FUNCTION "FC 141" : VOID	// FC 141
VERSION : 0.1
BEGIN
// (block stored without names or comments; labels and parameter names are numbered)
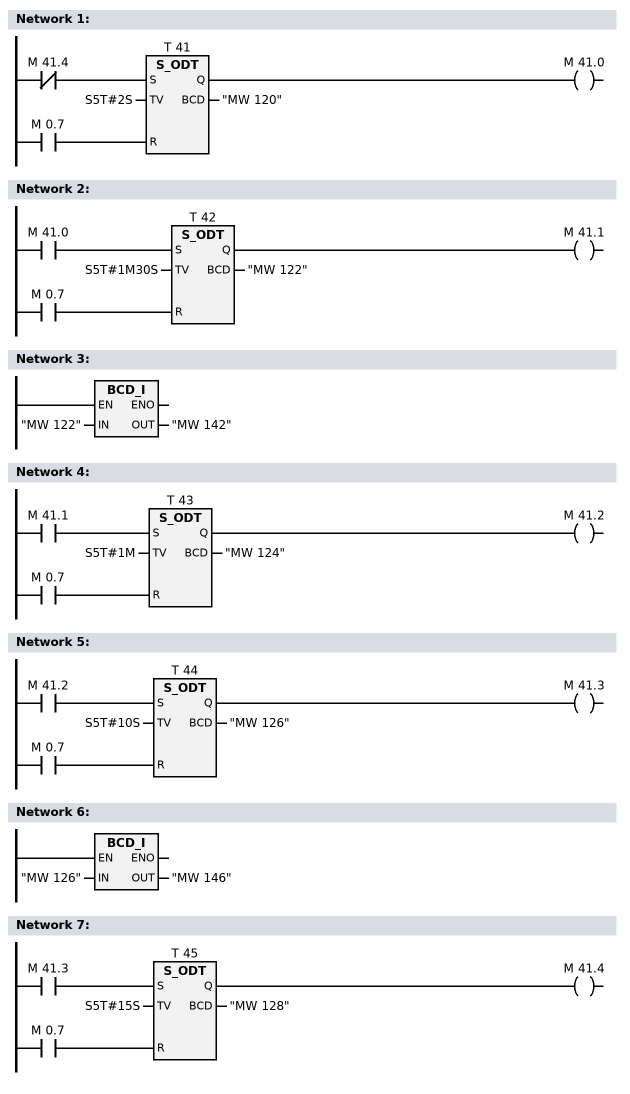
NETWORK
TITLE =
      AN    "M 41.4";
      L     S5T#2S;
      SD    "T 41";
      A     "M 0.7";
      R     "T 41";
      NOP   0;
      LC    "T 41";
      T     "MW 120";
      A     "T 41";
      =     "M 41.0";
NETWORK
TITLE =
      A     "M 41.0";
      L     S5T#1M30S;
      SD    "T 42";
      A     "M 0.7";
      R     "T 42";
      NOP   0;
      LC    "T 42";
      T     "MW 122";
      A     "T 42";
      =     "M 41.1";
NETWORK
TITLE =
      L     "MW 122";
      BTI;
      T     "MW 142";
      NOP   0;
NETWORK
TITLE =
      A     "M 41.1";
      L     S5T#1M;
      SD    "T 43";
      A     "M 0.7";
      R     "T 43";
      NOP   0;
      LC    "T 43";
      T     "MW 124";
      A     "T 43";
      =     "M 41.2";
NETWORK
TITLE =
      A     "M 41.2";
      L     S5T#10S;
      SD    "T 44";
      A     "M 0.7";
      R     "T 44";
      NOP   0;
      LC    "T 44";
      T     "MW 126";
      A     "T 44";
      =     "M 41.3";
NETWORK
TITLE =
      L     "MW 126";
      BTI;
      T     "MW 146";
      NOP   0;
NETWORK
TITLE =
      A     "M 41.3";
      L     S5T#15S;
      SD    "T 45";
      A     "M 0.7";
      R     "T 45";
      NOP   0;
      LC    "T 45";
      T     "MW 128";
      A     "T 45";
      =     "M 41.4";
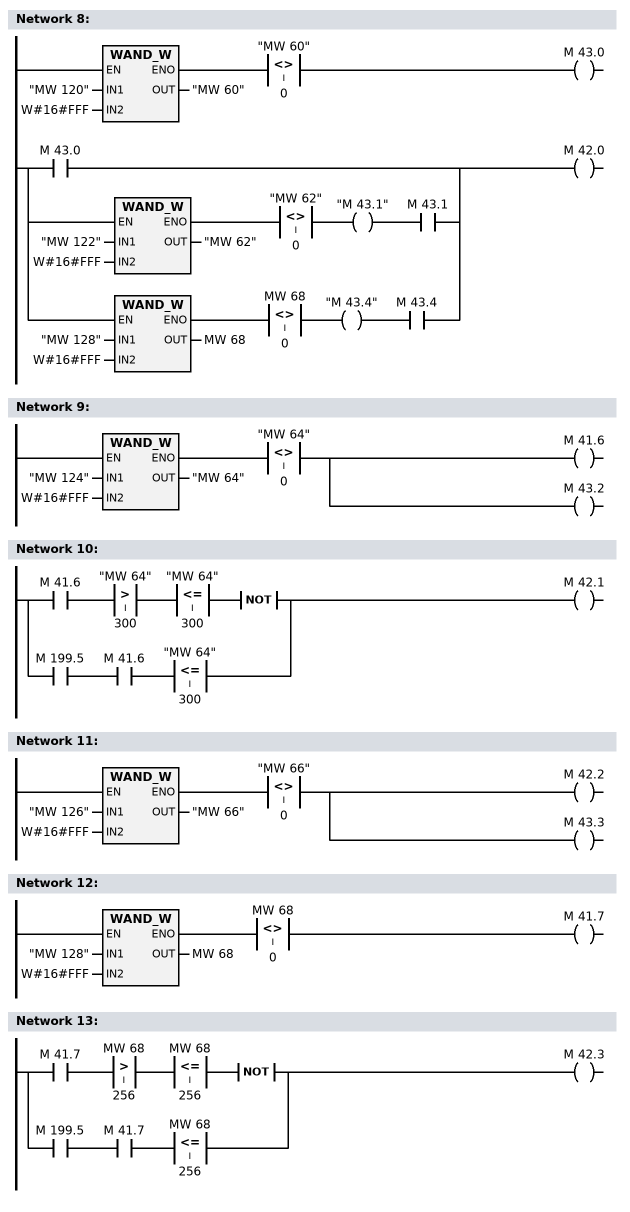
NETWORK
TITLE =
      A(;
      L     "MW 120";
      L     W#16#FFF;
      AW;
      T     "MW 60";
      SET;
      SAVE;
      CLR;
      A     BR;
      );
      A(;
      L     "MW 60";
      L     0;
      <>I;
      );
      =     "M 43.0";
      A     "M 43.0";
      O(;
      A(;
      L     "MW 122";
      L     W#16#FFF;
      AW;
      T     "MW 62";
      SET;
      SAVE;
      CLR;
      A     BR;
      );
      A(;
      L     "MW 62";
      L     0;
      <>I;
      );
      =     "M 43.1";
      A     "M 43.1";
      );
      O(;
      A(;
      L     "MW 128";
      L     W#16#FFF;
      AW;
      T     MW 68;
      SET;
      SAVE;
      CLR;
      A     BR;
      );
      A(;
      L     MW 68;
      L     0;
      <>I;
      );
      =     "M 43.4";
      A     "M 43.4";
      );
      =     "M 42.0";
NETWORK
TITLE =
      A(;
      L     "MW 124";
      L     W#16#FFF;
      AW;
      T     "MW 64";
      SET;
      SAVE;
      CLR;
      A     BR;
      );
      A(;
      L     "MW 64";
      L     0;
      <>I;
      );
      =     "M 41.6";
      =     "M 43.2";
NETWORK
TITLE =
      A     "M 41.6";
      A(;
      L     "MW 64";
      L     300;
      >I;
      );
      A(;
      A(;
      L     "MW 64";
      L     300;
      <=I;
      );
      NOT;
      );
      O;
      A     "M 199.5";
      A     "M 41.6";
      A(;
      L     "MW 64";
      L     300;
      <=I;
      );
      =     "M 42.1";
NETWORK
TITLE =
      A(;
      L     "MW 126";
      L     W#16#FFF;
      AW;
      T     "MW 66";
      SET;
      SAVE;
      CLR;
      A     BR;
      );
      A(;
      L     "MW 66";
      L     0;
      <>I;
      );
      =     "M 42.2";
      =     "M 43.3";
NETWORK
TITLE =
      A(;
      L     "MW 128";
      L     W#16#FFF;
      AW;
      T     MW 68;
      SET;
      SAVE;
      CLR;
      A     BR;
      );
      A(;
      L     MW 68;
      L     0;
      <>I;
      );
      =     "M 41.7";
NETWORK
TITLE =
      A     "M 41.7";
      A(;
      L     MW 68;
      L     256;
      >I;
      );
      A(;
      A(;
      L     MW 68;
      L     256;
      <=I;
      );
      NOT;
      );
      O;
      A     "M 199.5";
      A     "M 41.7";
      A(;
      L     MW 68;
      L     256;
      <=I;
      );
      =     "M 42.3";
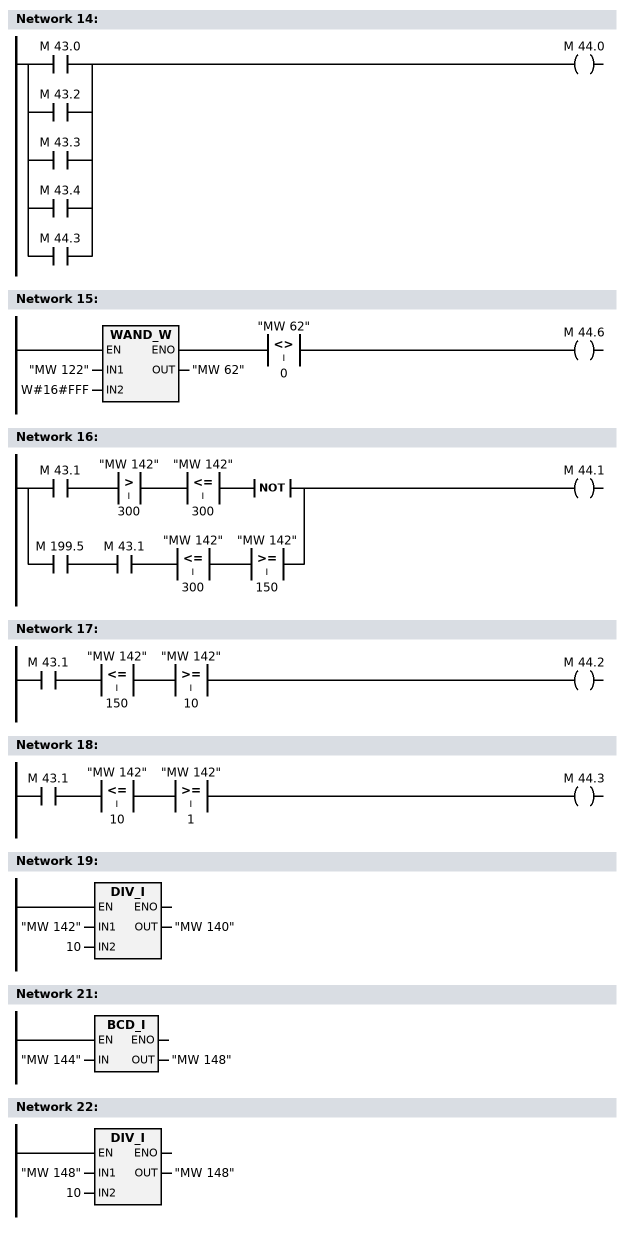
NETWORK
TITLE =
      O     "M 43.0";
      O     "M 43.2";
      O     "M 43.3";
      O     "M 43.4";
      O     M 44.3;
      =     "M 44.0";
NETWORK
TITLE =
      A(;
      L     "MW 122";
      L     W#16#FFF;
      AW;
      T     "MW 62";
      SET;
      SAVE;
      CLR;
      A     BR;
      );
      A(;
      L     "MW 62";
      L     0;
      <>I;
      );
      =     "M 44.6";
NETWORK
TITLE =
      A     "M 43.1";
      A(;
      L     "MW 142";
      L     300;
      >I;
      );
      A(;
      A(;
      L     "MW 142";
      L     300;
      <=I;
      );
      NOT;
      );
      O;
      A     "M 199.5";
      A     "M 43.1";
      A(;
      L     "MW 142";
      L     300;
      <=I;
      );
      A(;
      L     "MW 142";
      L     150;
      >=I;
      );
      =     "M 44.1";
NETWORK
TITLE =
      A     "M 43.1";
      A(;
      L     "MW 142";
      L     150;
      <=I;
      );
      A(;
      L     "MW 142";
      L     10;
      >=I;
      );
      =     "M 44.2";
NETWORK
TITLE =
      A     "M 43.1";
      A(;
      L     "MW 142";
      L     10;
      <=I;
      );
      A(;
      L     "MW 142";
      L     1;
      >=I;
      );
      =     M 44.3;
NETWORK
TITLE =
      L     "MW 142";
      L     10;
      /I;
      T     "MW 140";
      NOP   0;
NETWORK
TITLE =
      A(;
      A     "M 44.0";
      S     M 43.7;
      A     M 44.3;
      R     M 43.7;
      A     M 43.7;
      );
      L     S5T#1M10S;
      SD    "T 46";
      NOP   0;
      NOP   0;
      LC    "T 46";
      T     "MW 144";
      NOP   0;
NETWORK
TITLE =
      L     "MW 144";
      BTI;
      T     "MW 148";
      NOP   0;
NETWORK
TITLE =
      L     "MW 148";
      L     10;
      /I;
      T     "MW 148";
      NOP   0;
END_FUNCTION

FUNCTION "FC 142" : VOID	// FC 142
VERSION : 0.1
BEGIN
// (block stored without names or comments; labels and parameter names are numbered)
NETWORK
TITLE =
      A     "M 139.0";
      A     "M 139.1";
      CU    "Z 100";
      BLD   101;
      NOP   0;
      NOP   0;
      A(;
      L     "MW 150";
      L     60;
      >=I;
      );
      R     "Z 100";
      NOP   0;
      LC    "Z 100";
      T     "MW 160";
      NOP   0;
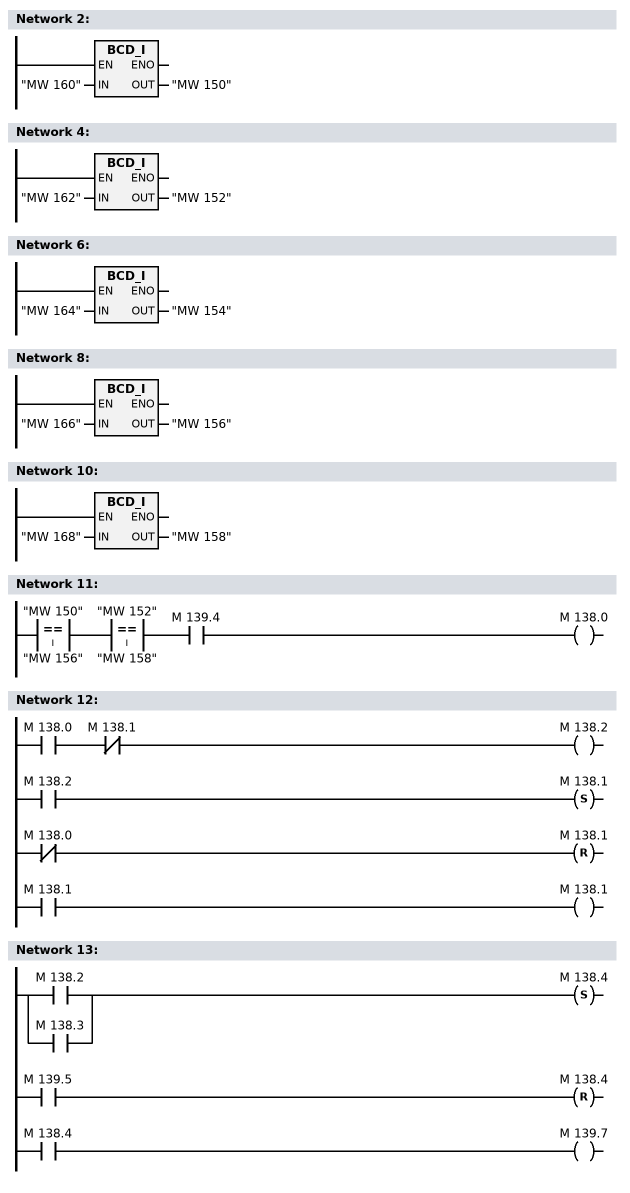
NETWORK
TITLE =
      L     "MW 160";
      BTI;
      T     "MW 150";
      NOP   0;
NETWORK
TITLE =
      A     "M 139.0";
      A     "M 139.2";
      CU    "Z 101";
      BLD   101;
      NOP   0;
      NOP   0;
      A(;
      L     "MW 152";
      L     24;
      >=I;
      );
      R     "Z 101";
      NOP   0;
      LC    "Z 101";
      T     "MW 162";
      NOP   0;
NETWORK
TITLE =
      L     "MW 162";
      BTI;
      T     "MW 152";
      NOP   0;
NETWORK
TITLE =
      A     "M 199.5";
      CU    "Z 102";
      BLD   101;
      NOP   0;
      NOP   0;
      A(;
      L     "MW 154";
      L     60;
      >=I;
      );
      R     "Z 102";
      NOP   0;
      LC    "Z 102";
      T     "MW 164";
      NOP   0;
NETWORK
TITLE =
      L     "MW 164";
      BTI;
      T     "MW 154";
      NOP   0;
NETWORK
TITLE =
      A(;
      A     "M 139.3";
      A     "M 139.1";
      O;
      A(;
      L     "MW 154";
      L     60;
      >=I;
      );
      AN    "M 139.3";
      );
      CU    "Z 103";
      BLD   101;
      NOP   0;
      NOP   0;
      A(;
      L     "MW 156";
      L     60;
      >=I;
      );
      R     "Z 103";
      NOP   0;
      LC    "Z 103";
      T     "MW 166";
      NOP   0;
NETWORK
TITLE =
      L     "MW 166";
      BTI;
      T     "MW 156";
      NOP   0;
NETWORK
TITLE =
      A(;
      A     "M 139.3";
      A     "M 139.2";
      O;
      A(;
      L     "MW 156";
      L     60;
      >=I;
      );
      AN    "M 139.3";
      );
      CU    "Z 104";
      BLD   101;
      NOP   0;
      NOP   0;
      A(;
      L     "MW 158";
      L     24;
      >=I;
      );
      R     "Z 104";
      NOP   0;
      LC    "Z 104";
      T     "MW 168";
      NOP   0;
NETWORK
TITLE =
      L     "MW 168";
      BTI;
      T     "MW 158";
      NOP   0;
NETWORK
TITLE =
      A(;
      L     "MW 150";
      L     "MW 156";
      ==I;
      );
      A(;
      L     "MW 152";
      L     "MW 158";
      ==I;
      );
      A     "M 139.4";
      =     "M 138.0";
NETWORK
TITLE =
      A     "M 138.0";
      AN    "M 138.1";
      =     "M 138.2";
      A     "M 138.2";
      S     "M 138.1";
      AN    "M 138.0";
      R     "M 138.1";
      A     "M 138.1";
      =     "M 138.1";
NETWORK
TITLE =
      A(;
      O     "M 138.2";
      O     "M 138.3";
      );
      S     "M 138.4";
      A     "M 139.5";
      R     "M 138.4";
      A     "M 138.4";
      =     "M 139.7";
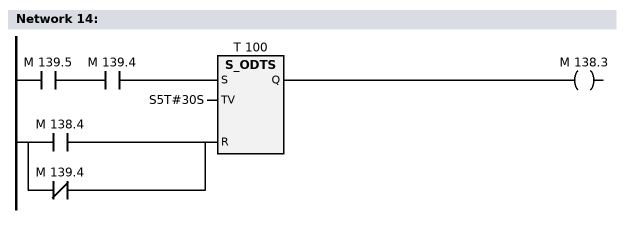
NETWORK
TITLE =
      A     "M 139.5";
      A     "M 139.4";
      L     S5T#30S;
      SS    "T 100";
      A(;
      O     "M 138.4";
      ON    "M 139.4";
      );
      R     "T 100";
      NOP   0;
      NOP   0;
      A     "T 100";
      =     "M 138.3";
END_FUNCTION

FUNCTION "FC 143" : VOID	// FC 143
VERSION : 0.1
BEGIN
// (block stored without names or comments; labels and parameter names are numbered)
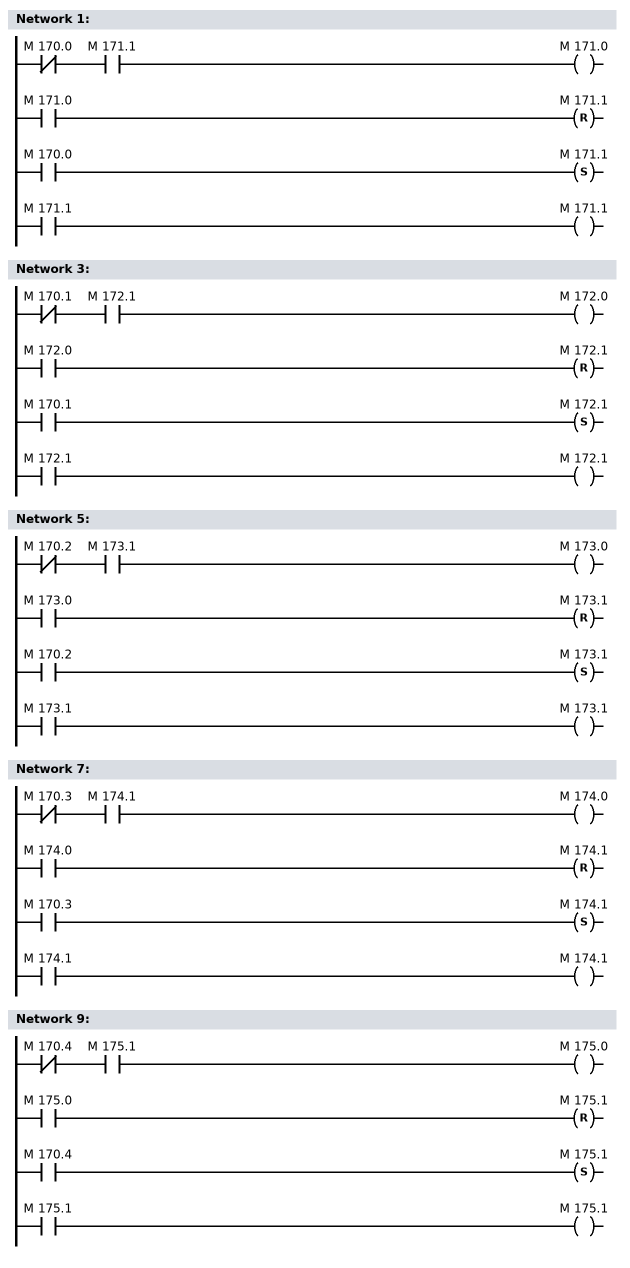
NETWORK
TITLE =
      AN    "M 170.0";
      A     "M 171.1";
      =     "M 171.0";
      A     "M 171.0";
      R     "M 171.1";
      A     "M 170.0";
      S     "M 171.1";
      A     "M 171.1";
      =     "M 171.1";
NETWORK
TITLE =
      A(;
      A     "M 171.0";
      S     "M 171.2";
      A     "M 190.1";
      R     "M 171.2";
      A     "M 171.2";
      );
      A     "M 1.5";
      O;
      AN    "M 171.2";
      A(;
      A     "M 171.0";
      S     "M 171.3";
      A     "M 190.2";
      A     "M 170.0";
      R     "M 171.3";
      A     "M 171.3";
      );
      O     "M 190.3";
      =     "M 171.4";
      =     "1H1";
NETWORK
TITLE =
      AN    "M 170.1";
      A     "M 172.1";
      =     "M 172.0";
      A     "M 172.0";
      R     "M 172.1";
      A     "M 170.1";
      S     "M 172.1";
      A     "M 172.1";
      =     "M 172.1";
NETWORK
TITLE =
      A(;
      A     "M 172.0";
      S     "M 172.2";
      A     "M 190.1";
      R     "M 172.2";
      A     "M 172.2";
      );
      A     "M 1.5";
      O;
      AN    "M 172.2";
      A(;
      A     "M 172.0";
      S     "M 172.3";
      A     "M 190.2";
      A     "M 170.1";
      R     "M 172.3";
      A     "M 172.3";
      );
      O     "M 190.3";
      =     "M 172.4";
      =     "2H1";
NETWORK
TITLE =
      AN    "M 170.2";
      A     "M 173.1";
      =     "M 173.0";
      A     "M 173.0";
      R     "M 173.1";
      A     "M 170.2";
      S     "M 173.1";
      A     "M 173.1";
      =     "M 173.1";
NETWORK
TITLE =
      A(;
      A     "M 173.0";
      S     "M 173.2";
      A     "M 190.1";
      R     "M 173.2";
      A     "M 173.2";
      );
      A     "M 1.5";
      O;
      AN    "M 173.2";
      A(;
      A     "M 173.0";
      S     "M 173.3";
      A     "M 190.2";
      A     "M 170.2";
      R     "M 173.3";
      A     "M 173.3";
      );
      O     "M 190.3";
      =     "M 173.4";
      =     "3H1";
NETWORK
TITLE =
      AN    "M 170.3";
      A     "M 174.1";
      =     "M 174.0";
      A     "M 174.0";
      R     "M 174.1";
      A     "M 170.3";
      S     "M 174.1";
      A     "M 174.1";
      =     "M 174.1";
NETWORK
TITLE =
      A(;
      A     "M 174.0";
      S     "M 174.2";
      A     "M 190.1";
      R     "M 174.2";
      A     "M 174.2";
      );
      A     "M 1.5";
      O;
      AN    "M 174.2";
      A(;
      A     "M 174.0";
      S     "M 174.3";
      A     "M 190.2";
      A     "M 170.3";
      R     "M 174.3";
      A     "M 174.3";
      );
      O     "M 190.3";
      =     "M 174.4";
      =     "4H1";
NETWORK
TITLE =
      AN    "M 170.4";
      A     "M 175.1";
      =     "M 175.0";
      A     "M 175.0";
      R     "M 175.1";
      A     "M 170.4";
      S     "M 175.1";
      A     "M 175.1";
      =     "M 175.1";
NETWORK
TITLE =
      A(;
      A     "M 175.0";
      S     "M 175.2";
      A     "M 190.1";
      R     "M 175.2";
      A     "M 175.2";
      );
      A     "M 1.5";
      O;
      AN    "M 175.2";
      A(;
      A     "M 175.0";
      S     "M 175.3";
      A     "M 190.2";
      A     "M 170.4";
      R     "M 175.3";
      A     "M 175.3";
      );
      O     "M 190.3";
      =     "M 175.4";
      =     "5H1";
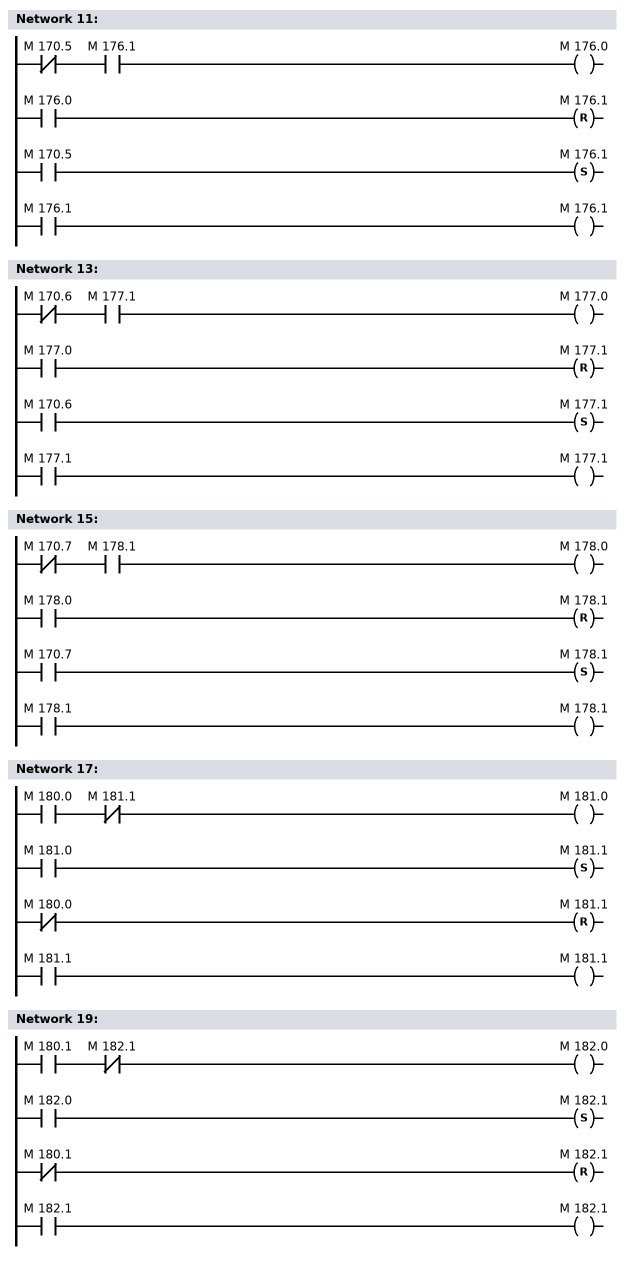
NETWORK
TITLE =
      AN    "M 170.5";
      A     "M 176.1";
      =     "M 176.0";
      A     "M 176.0";
      R     "M 176.1";
      A     "M 170.5";
      S     "M 176.1";
      A     "M 176.1";
      =     "M 176.1";
NETWORK
TITLE =
      A(;
      A     "M 176.0";
      S     "M 176.2";
      A     "M 190.1";
      R     "M 176.2";
      A     "M 176.2";
      );
      A     "M 1.5";
      O;
      AN    "M 176.2";
      A(;
      A     "M 176.0";
      S     "M 176.3";
      A     "M 190.2";
      A     "M 170.5";
      R     "M 176.3";
      A     "M 176.3";
      );
      O     "M 190.3";
      =     "M 176.4";
      =     "6H1";
NETWORK
TITLE =
      AN    "M 170.6";
      A     "M 177.1";
      =     "M 177.0";
      A     "M 177.0";
      R     "M 177.1";
      A     "M 170.6";
      S     "M 177.1";
      A     "M 177.1";
      =     "M 177.1";
NETWORK
TITLE =
      A(;
      A     "M 177.0";
      S     "M 177.2";
      A     "M 190.1";
      R     "M 177.2";
      A     "M 177.2";
      );
      A     "M 1.5";
      O;
      AN    "M 177.2";
      A(;
      A     "M 177.0";
      S     "M 177.3";
      A     "M 190.2";
      A     "M 170.6";
      R     "M 177.3";
      A     "M 177.3";
      );
      O     "M 190.3";
      =     "M 177.4";
      =     "7H1";
NETWORK
TITLE =
      AN    "M 170.7";
      A     "M 178.1";
      =     "M 178.0";
      A     "M 178.0";
      R     "M 178.1";
      A     "M 170.7";
      S     "M 178.1";
      A     "M 178.1";
      =     "M 178.1";
NETWORK
TITLE =
      A(;
      A     "M 178.0";
      S     "M 178.2";
      A     "M 190.1";
      R     "M 178.2";
      A     "M 178.2";
      );
      A     "M 1.5";
      O;
      AN    "M 178.2";
      A(;
      A     "M 178.0";
      S     "M 178.3";
      A     "M 190.2";
      A     "M 170.7";
      R     "M 178.3";
      A     "M 178.3";
      );
      O     "M 190.3";
      =     "M 178.4";
      =     "8H1";
NETWORK
TITLE =
      A     "M 180.0";
      AN    "M 181.1";
      =     "M 181.0";
      A     "M 181.0";
      S     "M 181.1";
      AN    "M 180.0";
      R     "M 181.1";
      A     "M 181.1";
      =     "M 181.1";
NETWORK
TITLE =
      A(;
      A     "M 181.0";
      S     "M 181.2";
      A     "M 190.1";
      R     "M 181.2";
      A     "M 181.2";
      );
      A     "M 1.5";
      O;
      AN    "M 181.2";
      A(;
      A     "M 181.0";
      S     "M 181.3";
      A     "M 190.2";
      AN    "M 180.0";
      R     "M 181.3";
      A     "M 181.3";
      );
      O     "M 190.3";
      =     "M 181.4";
      =     "1H2";
NETWORK
TITLE =
      A     "M 180.1";
      AN    "M 182.1";
      =     "M 182.0";
      A     "M 182.0";
      S     "M 182.1";
      AN    "M 180.1";
      R     "M 182.1";
      A     "M 182.1";
      =     "M 182.1";
NETWORK
TITLE =
      A(;
      A     "M 182.0";
      S     "M 182.2";
      A     "M 190.1";
      R     "M 182.2";
      A     "M 182.2";
      );
      A     "M 1.5";
      O;
      AN    "M 182.2";
      A(;
      A     "M 182.0";
      S     "M 182.3";
      A     "M 190.2";
      AN    "M 180.1";
      R     "M 182.3";
      A     "M 182.3";
      );
      O     "M 190.3";
      =     "M 182.4";
      =     "2H2";
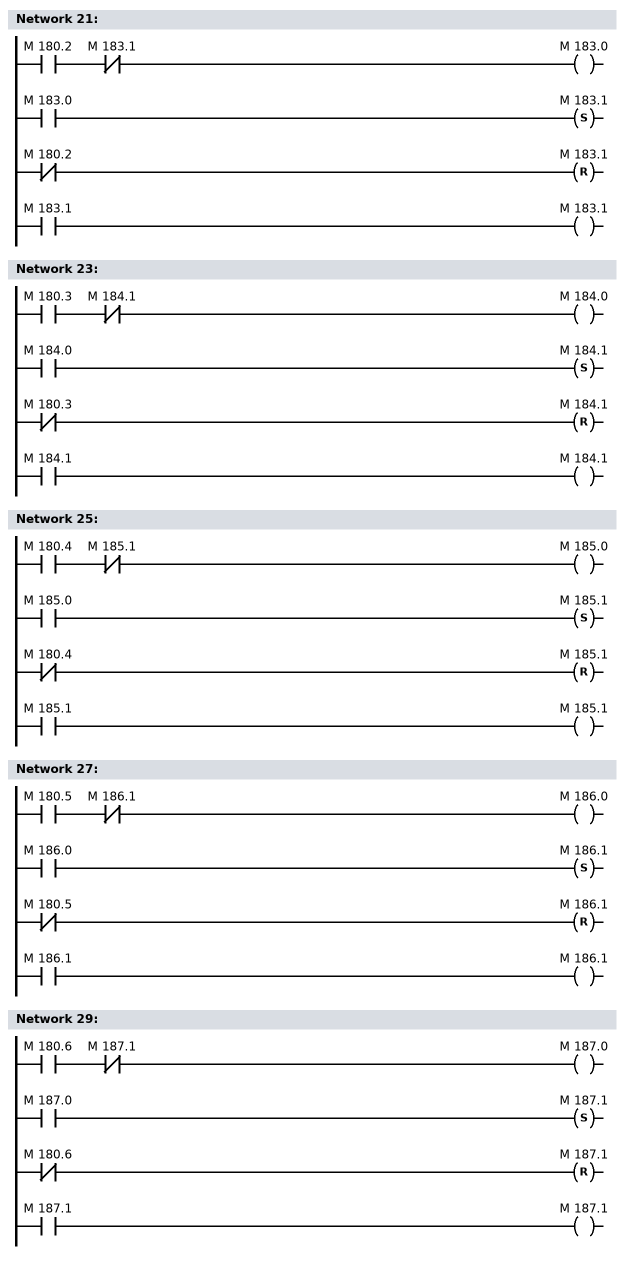
NETWORK
TITLE =
      A     "M 180.2";
      AN    "M 183.1";
      =     "M 183.0";
      A     "M 183.0";
      S     "M 183.1";
      AN    "M 180.2";
      R     "M 183.1";
      A     "M 183.1";
      =     "M 183.1";
NETWORK
TITLE =
      A(;
      A     "M 183.0";
      S     "M 183.2";
      A     "M 190.1";
      R     "M 183.2";
      A     "M 183.2";
      );
      A     "M 1.5";
      O;
      AN    "M 183.2";
      A(;
      A     "M 183.0";
      S     "M 183.3";
      A     "M 190.2";
      AN    "M 180.2";
      R     "M 183.3";
      A     "M 183.3";
      );
      O     "M 190.3";
      =     "M 183.4";
      =     "3H2";
NETWORK
TITLE =
      A     "M 180.3";
      AN    "M 184.1";
      =     "M 184.0";
      A     "M 184.0";
      S     "M 184.1";
      AN    "M 180.3";
      R     "M 184.1";
      A     "M 184.1";
      =     "M 184.1";
NETWORK
TITLE =
      A(;
      A     "M 184.0";
      S     "M 184.2";
      A     "M 190.1";
      R     "M 184.2";
      A     "M 184.2";
      );
      A     "M 1.5";
      O;
      AN    "M 184.2";
      A(;
      A     "M 184.0";
      S     "M 184.3";
      A     "M 190.2";
      AN    "M 180.3";
      R     "M 184.3";
      A     "M 184.3";
      );
      O     "M 190.3";
      =     "M 184.4";
      =     "4H2";
NETWORK
TITLE =
      A     "M 180.4";
      AN    "M 185.1";
      =     "M 185.0";
      A     "M 185.0";
      S     "M 185.1";
      AN    "M 180.4";
      R     "M 185.1";
      A     "M 185.1";
      =     "M 185.1";
NETWORK
TITLE =
      A(;
      A     "M 185.0";
      S     "M 185.2";
      A     "M 190.1";
      R     "M 185.2";
      A     "M 185.2";
      );
      A     "M 1.5";
      O;
      AN    "M 185.2";
      A(;
      A     "M 185.0";
      S     "M 185.3";
      A     "M 190.2";
      AN    "M 180.4";
      R     "M 185.3";
      A     "M 185.3";
      );
      O     "M 190.3";
      =     "M 185.4";
      =     "5H2";
NETWORK
TITLE =
      A     "M 180.5";
      AN    "M 186.1";
      =     "M 186.0";
      A     "M 186.0";
      S     "M 186.1";
      AN    "M 180.5";
      R     "M 186.1";
      A     "M 186.1";
      =     "M 186.1";
NETWORK
TITLE =
      A(;
      A     "M 186.0";
      S     "M 186.2";
      A     "M 190.1";
      R     "M 186.2";
      A     "M 186.2";
      );
      A     "M 1.5";
      O;
      AN    "M 186.2";
      A(;
      A     "M 186.0";
      S     "M 186.3";
      A     "M 190.2";
      AN    "M 180.5";
      R     "M 186.3";
      A     "M 186.3";
      );
      O     "M 190.3";
      =     "M 186.4";
      =     "6H2";
NETWORK
TITLE =
      A     "M 180.6";
      AN    "M 187.1";
      =     "M 187.0";
      A     "M 187.0";
      S     "M 187.1";
      AN    "M 180.6";
      R     "M 187.1";
      A     "M 187.1";
      =     "M 187.1";
NETWORK
TITLE =
      A(;
      A     "M 187.0";
      S     "M 187.2";
      A     "M 190.1";
      R     "M 187.2";
      A     "M 187.2";
      );
      A     "M 1.5";
      O;
      AN    "M 187.2";
      A(;
      A     "M 187.0";
      S     "M 187.3";
      A     "M 190.2";
      AN    "M 180.6";
      R     "M 187.3";
      A     "M 187.3";
      );
      O     "M 190.3";
      =     "M 187.4";
      =     "7H2";
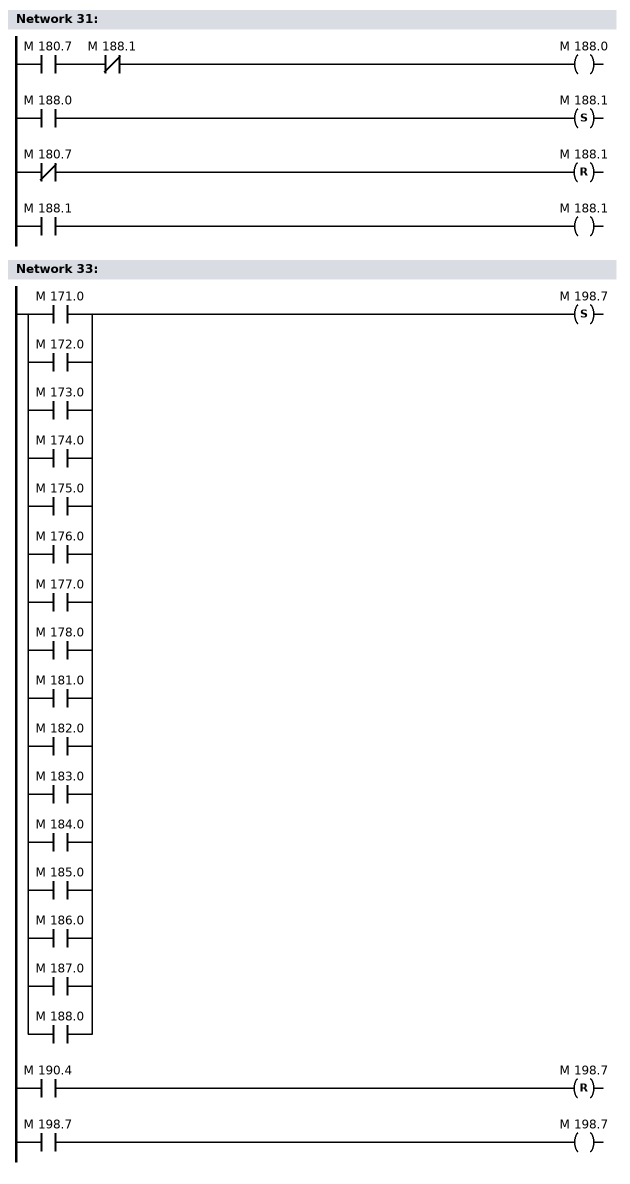
NETWORK
TITLE =
      A     "M 180.7";
      AN    "M 188.1";
      =     "M 188.0";
      A     "M 188.0";
      S     "M 188.1";
      AN    "M 180.7";
      R     "M 188.1";
      A     "M 188.1";
      =     "M 188.1";
NETWORK
TITLE =
      A(;
      A     "M 188.0";
      S     "M 188.2";
      A     "M 190.1";
      R     "M 188.2";
      A     "M 188.2";
      );
      A     "M 1.5";
      O;
      AN    "M 188.2";
      A(;
      A     "M 188.0";
      S     "M 188.3";
      A     "M 190.2";
      AN    "M 180.7";
      R     "M 188.3";
      A     "M 188.3";
      );
      O     "M 190.3";
      =     "M 188.4";
      =     "8H2";
NETWORK
TITLE =
      A(;
      O     "M 171.0";
      O     "M 172.0";
      O     "M 173.0";
      O     "M 174.0";
      O     "M 175.0";
      O     "M 176.0";
      O     "M 177.0";
      O     "M 178.0";
      O     "M 181.0";
      O     "M 182.0";
      O     "M 183.0";
      O     "M 184.0";
      O     "M 185.0";
      O     "M 186.0";
      O     "M 187.0";
      O     "M 188.0";
      );
      S     "M 198.7";
      A     "M 190.4";
      R     "M 198.7";
      A     "M 198.7";
      =     "M 198.7";
END_FUNCTION

FUNCTION "FC 160" : VOID	// FC 160
VERSION : 0.1
BEGIN
// (block stored without names or comments; labels and parameter names are numbered)
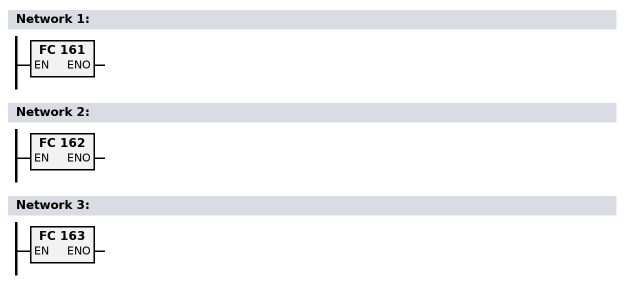
NETWORK
TITLE =
      CALL  "FC 161";
      NOP   0;
NETWORK
TITLE =
      CALL  "FC 162";
      NOP   0;
NETWORK
TITLE =
      CALL  "FC 163";
      NOP   0;
END_FUNCTION

FUNCTION "FC 161" : VOID	// FC 161
VERSION : 0.1
BEGIN
// (block stored without names or comments; labels and parameter names are numbered)
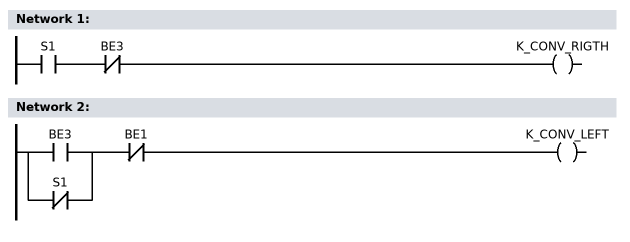
NETWORK
TITLE =
      A     "S1";
      AN    "BE3";
      =     "K_CONV_RIGTH";
NETWORK
TITLE =
      A(;
      O     "BE3";
      ON    "S1";
      );
      AN    "BE1";
      =     "K_CONV_LEFT";
END_FUNCTION

FUNCTION "FC 162" : VOID	// FC 162
VERSION : 0.1
BEGIN
// (block stored without names or comments; labels and parameter names are numbered)
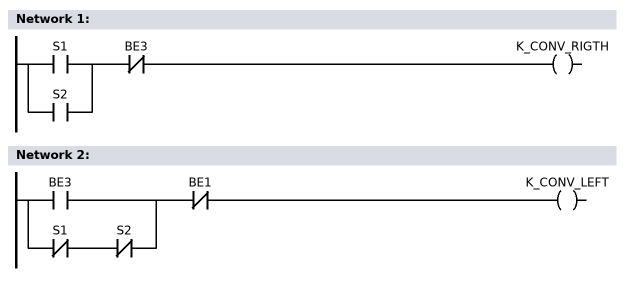
NETWORK
TITLE =
      A(;
      O     "S1";
      O     "S2";
      );
      AN    "BE3";
      =     "K_CONV_RIGTH";
NETWORK
TITLE =
      A(;
      O     "BE3";
      O;
      AN    "S1";
      AN    "S2";
      );
      AN    "BE1";
      =     "K_CONV_LEFT";
END_FUNCTION

FUNCTION "FC 163" : VOID	// FC 163
VERSION : 0.1
BEGIN
// (block stored without names or comments; labels and parameter names are numbered)
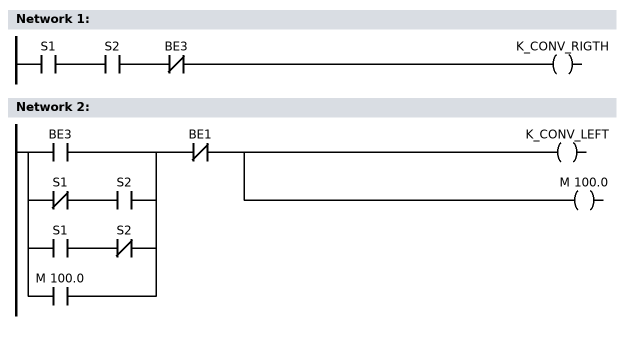
NETWORK
TITLE =
      A     "S1";
      A     "S2";
      AN    "BE3";
      =     "K_CONV_RIGTH";
NETWORK
TITLE =
      A(;
      O     "BE3";
      O;
      AN    "S1";
      A     "S2";
      O;
      A     "S1";
      AN    "S2";
      O     M 100.0;
      );
      AN    "BE1";
      =     "K_CONV_LEFT";
      =     M 100.0;
END_FUNCTION

FUNCTION "FC 164" : VOID	// FC 164
VERSION : 0.1
BEGIN
// (block stored without names or comments; labels and parameter names are numbered)
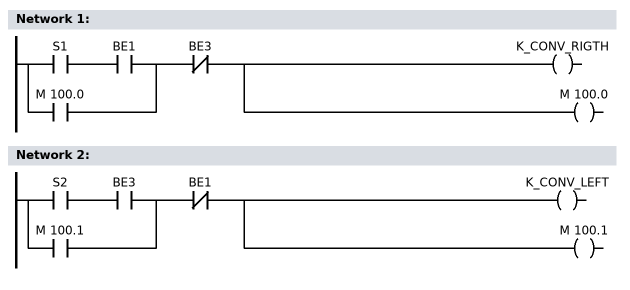
NETWORK
TITLE =
      A(;
      A     "S1";
      A     "BE1";
      O     M 100.0;
      );
      AN    "BE3";
      =     "K_CONV_RIGTH";
      =     M 100.0;
NETWORK
TITLE =
      A(;
      A     "S2";
      A     "BE3";
      O     M 100.1;
      );
      AN    "BE1";
      =     "K_CONV_LEFT";
      =     M 100.1;
END_FUNCTION

FUNCTION "FC 165" : VOID	// FC 165
VERSION : 0.1
BEGIN
// (block stored without names or comments; labels and parameter names are numbered)
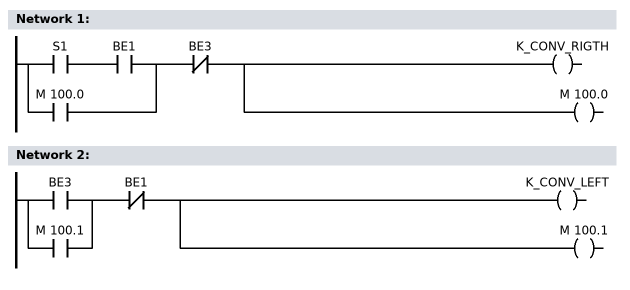
NETWORK
TITLE =
      A(;
      A     "S1";
      A     "BE1";
      O     M 100.0;
      );
      AN    "BE3";
      =     "K_CONV_RIGTH";
      =     M 100.0;
NETWORK
TITLE =
      A(;
      O     "BE3";
      O     M 100.1;
      );
      AN    "BE1";
      =     "K_CONV_LEFT";
      =     M 100.1;
END_FUNCTION

FUNCTION "FC 166" : VOID	// FC 166
VERSION : 0.1
BEGIN
// (block stored without names or comments; labels and parameter names are numbered)
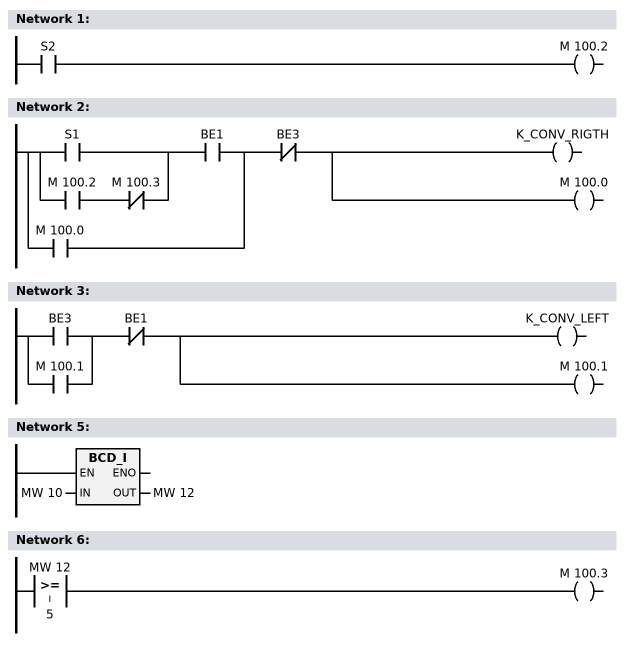
NETWORK
TITLE =
      A     "S2";
      =     M 100.2;
NETWORK
TITLE =
      A(;
      A(;
      O     "S1";
      O;
      A     M 100.2;
      AN    M 100.3;
      );
      A     "BE1";
      O     M 100.0;
      );
      AN    "BE3";
      =     "K_CONV_RIGTH";
      =     M 100.0;
NETWORK
TITLE =
      A(;
      O     "BE3";
      O     M 100.1;
      );
      AN    "BE1";
      =     "K_CONV_LEFT";
      =     M 100.1;
NETWORK
TITLE =
      A     "BE3";
      CU    "Z 1";
      BLD   101;
      NOP   0;
      NOP   0;
      AN    M 100.2;
      R     "Z 1";
      NOP   0;
      LC    "Z 1";
      T     MW 10;
      NOP   0;
NETWORK
TITLE =
      L     MW 10;
      BTI;
      T     MW 12;
      NOP   0;
NETWORK
TITLE =
      L     MW 12;
      L     5;
      >=I;
      =     M 100.3;
END_FUNCTION

FUNCTION "FC 167" : VOID	// FC 167
VERSION : 0.1
BEGIN
// (block stored without names or comments; labels and parameter names are numbered)
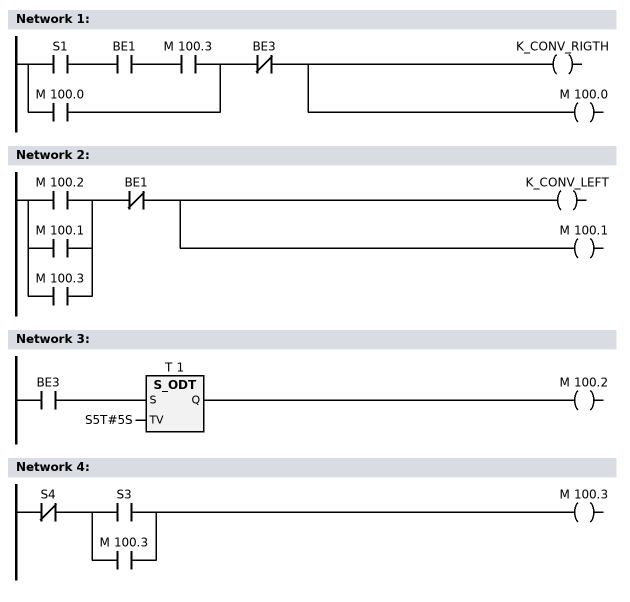
NETWORK
TITLE =
      A(;
      A     "S1";
      A     "BE1";
      A     M 100.3;
      O     M 100.0;
      );
      AN    "BE3";
      =     "K_CONV_RIGTH";
      =     M 100.0;
NETWORK
TITLE =
      A(;
      O     M 100.2;
      O     M 100.1;
      O     M 100.3;
      );
      AN    "BE1";
      =     "K_CONV_LEFT";
      =     M 100.1;
NETWORK
TITLE =
      A     "BE3";
      L     S5T#5S;
      SD    "T 1";
      NOP   0;
      NOP   0;
      NOP   0;
      A     "T 1";
      =     M 100.2;
NETWORK
TITLE =
      AN    "S4";
      A(;
      O     "S3";
      O     M 100.3;
      );
      =     M 100.3;
END_FUNCTION

FUNCTION "FC 240" : VOID	// FC 240
VERSION : 0.1
BEGIN
// (block stored without names or comments; labels and parameter names are numbered)
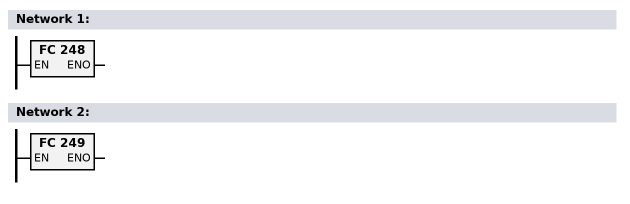
NETWORK
TITLE =
      CALL  "FC 248";
      NOP   0;
NETWORK
TITLE =
      CALL  "FC 249";
      NOP   0;
END_FUNCTION

FUNCTION "FC 248" : VOID	// FC 248
VERSION : 0.1
BEGIN
// (block stored without names or comments; labels and parameter names are numbered)
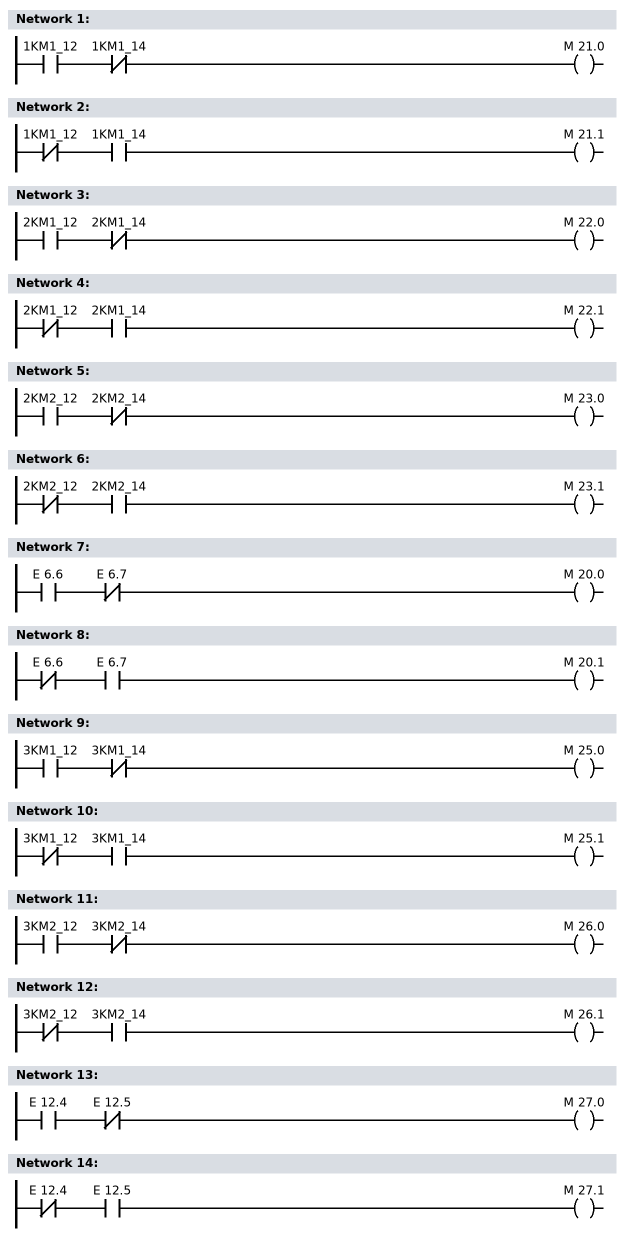
NETWORK
TITLE =
      A     "1KM1_12";
      AN    "1KM1_14";
      =     "M 21.0";
NETWORK
TITLE =
      AN    "1KM1_12";
      A     "1KM1_14";
      =     "M 21.1";
NETWORK
TITLE =
      A     "2KM1_12";
      AN    "2KM1_14";
      =     "M 22.0";
NETWORK
TITLE =
      AN    "2KM1_12";
      A     "2KM1_14";
      =     "M 22.1";
NETWORK
TITLE =
      A     "2KM2_12";
      AN    "2KM2_14";
      =     "M 23.0";
NETWORK
TITLE =
      AN    "2KM2_12";
      A     "2KM2_14";
      =     "M 23.1";
NETWORK
TITLE =
      A     "E 6.6";
      AN    "E 6.7";
      =     "M 20.0";
NETWORK
TITLE =
      AN    "E 6.6";
      A     "E 6.7";
      =     "M 20.1";
NETWORK
TITLE =
      A     "3KM1_12";
      AN    "3KM1_14";
      =     "M 25.0";
NETWORK
TITLE =
      AN    "3KM1_12";
      A     "3KM1_14";
      =     "M 25.1";
NETWORK
TITLE =
      A     "3KM2_12";
      AN    "3KM2_14";
      =     "M 26.0";
NETWORK
TITLE =
      AN    "3KM2_12";
      A     "3KM2_14";
      =     "M 26.1";
NETWORK
TITLE =
      A     "E 12.4";
      AN    "E 12.5";
      =     "M 27.0";
NETWORK
TITLE =
      AN    "E 12.4";
      A     "E 12.5";
      =     "M 27.1";
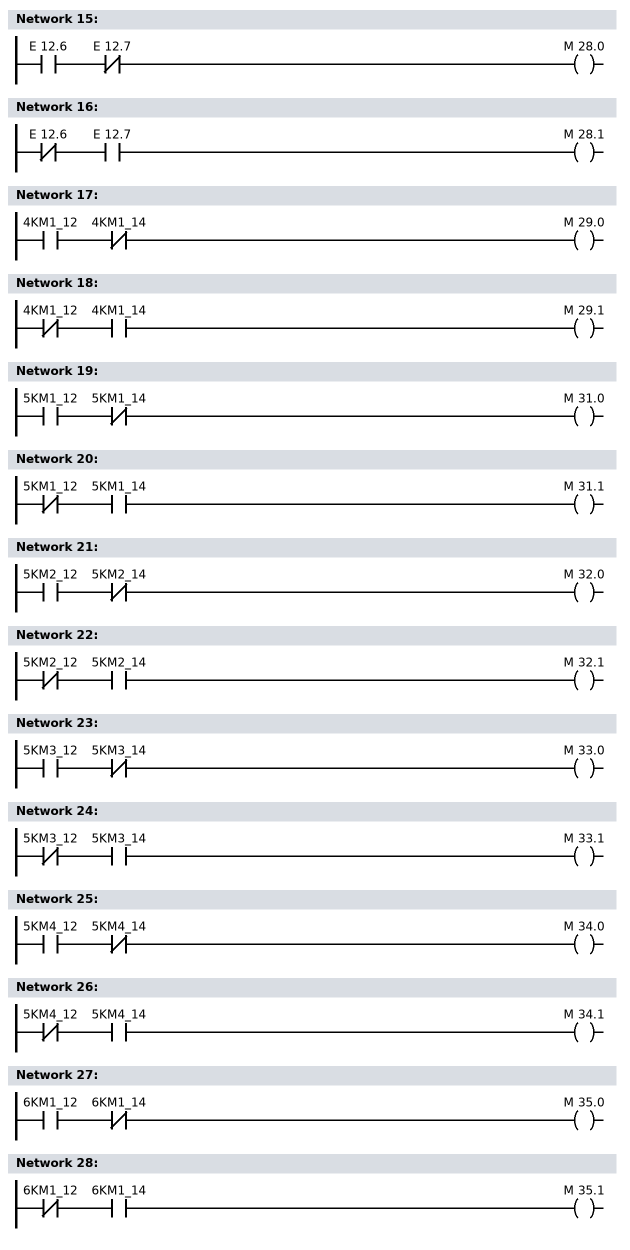
NETWORK
TITLE =
      A     "E 12.6";
      AN    "E 12.7";
      =     "M 28.0";
NETWORK
TITLE =
      AN    "E 12.6";
      A     "E 12.7";
      =     "M 28.1";
NETWORK
TITLE =
      A     "4KM1_12";
      AN    "4KM1_14";
      =     "M 29.0";
NETWORK
TITLE =
      AN    "4KM1_12";
      A     "4KM1_14";
      =     "M 29.1";
NETWORK
TITLE =
      A     "5KM1_12";
      AN    "5KM1_14";
      =     "M 31.0";
NETWORK
TITLE =
      AN    "5KM1_12";
      A     "5KM1_14";
      =     "M 31.1";
NETWORK
TITLE =
      A     "5KM2_12";
      AN    "5KM2_14";
      =     "M 32.0";
NETWORK
TITLE =
      AN    "5KM2_12";
      A     "5KM2_14";
      =     "M 32.1";
NETWORK
TITLE =
      A     "5KM3_12";
      AN    "5KM3_14";
      =     "M 33.0";
NETWORK
TITLE =
      AN    "5KM3_12";
      A     "5KM3_14";
      =     "M 33.1";
NETWORK
TITLE =
      A     "5KM4_12";
      AN    "5KM4_14";
      =     "M 34.0";
NETWORK
TITLE =
      AN    "5KM4_12";
      A     "5KM4_14";
      =     "M 34.1";
NETWORK
TITLE =
      A     "6KM1_12";
      AN    "6KM1_14";
      =     "M 35.0";
NETWORK
TITLE =
      AN    "6KM1_12";
      A     "6KM1_14";
      =     "M 35.1";
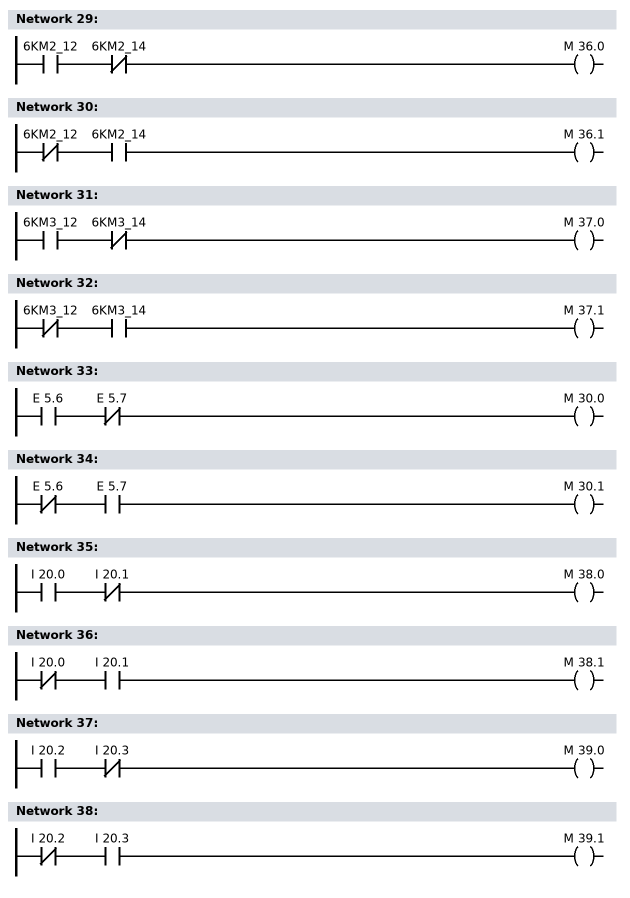
NETWORK
TITLE =
      A     "6KM2_12";
      AN    "6KM2_14";
      =     "M 36.0";
NETWORK
TITLE =
      AN    "6KM2_12";
      A     "6KM2_14";
      =     "M 36.1";
NETWORK
TITLE =
      A     "6KM3_12";
      AN    "6KM3_14";
      =     "M 37.0";
NETWORK
TITLE =
      AN    "6KM3_12";
      A     "6KM3_14";
      =     "M 37.1";
NETWORK
TITLE =
      A     "E 5.6";
      AN    "E 5.7";
      =     "M 30.0";
NETWORK
TITLE =
      AN    "E 5.6";
      A     "E 5.7";
      =     "M 30.1";
NETWORK
TITLE =
      A     I 20.0;
      AN    I 20.1;
      =     "M 38.0";
NETWORK
TITLE =
      AN    I 20.0;
      A     I 20.1;
      =     "M 38.1";
NETWORK
TITLE =
      A     I 20.2;
      AN    I 20.3;
      =     "M 39.0";
NETWORK
TITLE =
      AN    I 20.2;
      A     I 20.3;
      =     "M 39.1";
END_FUNCTION

FUNCTION "FC 249" : VOID	// FC 249
VERSION : 0.1
BEGIN
// (block stored without names or comments; labels and parameter names are numbered)
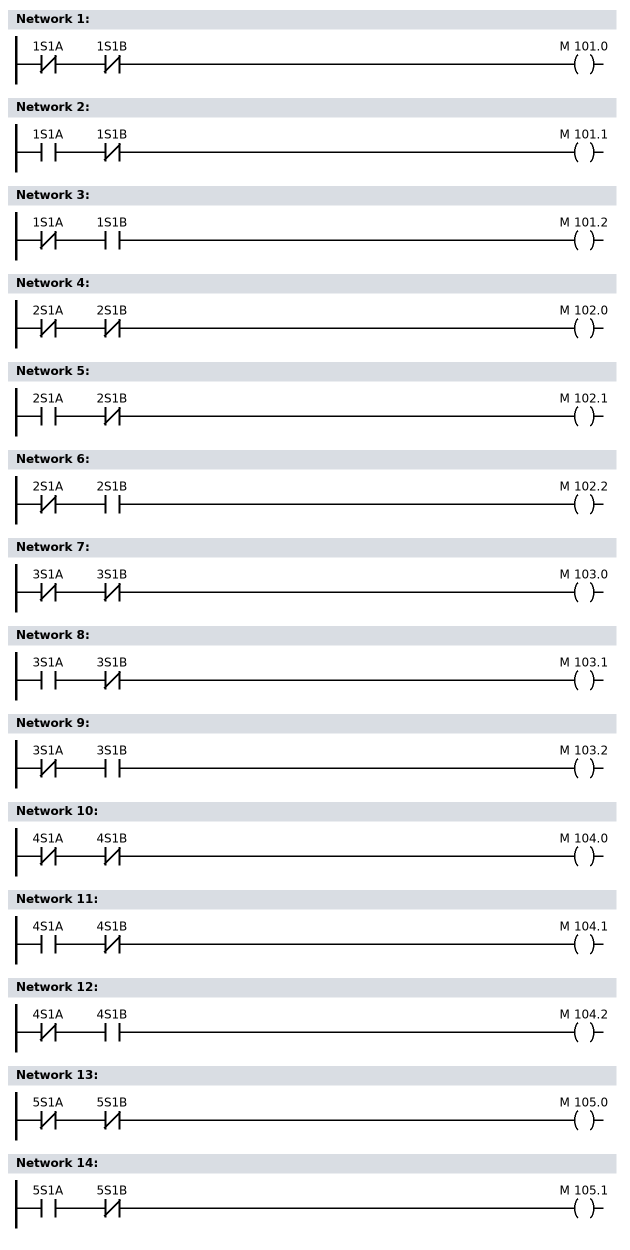
NETWORK
TITLE =
      AN    "1S1A";
      AN    "1S1B";
      =     "M 101.0";
NETWORK
TITLE =
      A     "1S1A";
      AN    "1S1B";
      =     "M 101.1";
NETWORK
TITLE =
      AN    "1S1A";
      A     "1S1B";
      =     "M 101.2";
NETWORK
TITLE =
      AN    "2S1A";
      AN    "2S1B";
      =     "M 102.0";
NETWORK
TITLE =
      A     "2S1A";
      AN    "2S1B";
      =     "M 102.1";
NETWORK
TITLE =
      AN    "2S1A";
      A     "2S1B";
      =     "M 102.2";
NETWORK
TITLE =
      AN    "3S1A";
      AN    "3S1B";
      =     "M 103.0";
NETWORK
TITLE =
      A     "3S1A";
      AN    "3S1B";
      =     "M 103.1";
NETWORK
TITLE =
      AN    "3S1A";
      A     "3S1B";
      =     "M 103.2";
NETWORK
TITLE =
      AN    "4S1A";
      AN    "4S1B";
      =     "M 104.0";
NETWORK
TITLE =
      A     "4S1A";
      AN    "4S1B";
      =     "M 104.1";
NETWORK
TITLE =
      AN    "4S1A";
      A     "4S1B";
      =     "M 104.2";
NETWORK
TITLE =
      AN    "5S1A";
      AN    "5S1B";
      =     "M 105.0";
NETWORK
TITLE =
      A     "5S1A";
      AN    "5S1B";
      =     "M 105.1";
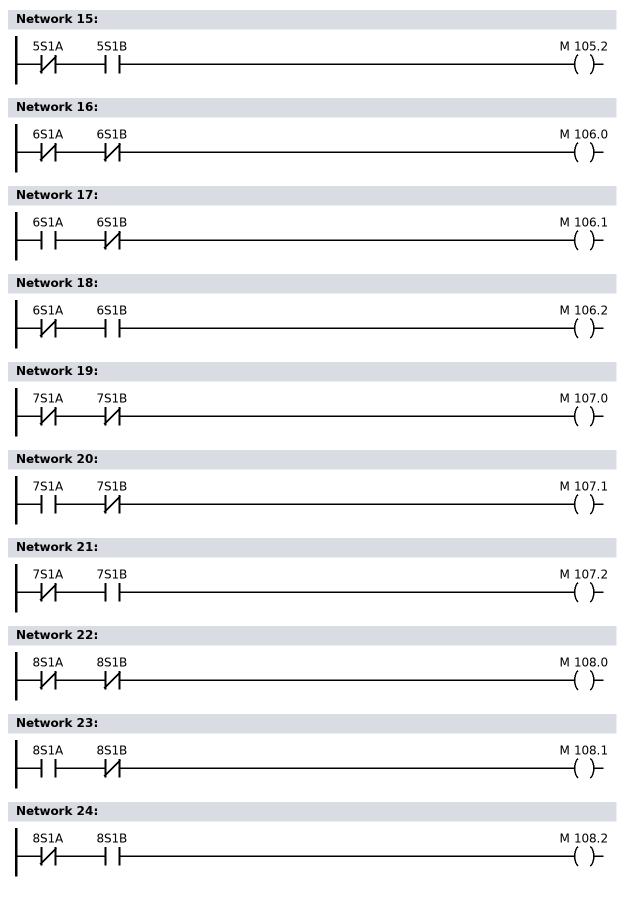
NETWORK
TITLE =
      AN    "5S1A";
      A     "5S1B";
      =     "M 105.2";
NETWORK
TITLE =
      AN    "6S1A";
      AN    "6S1B";
      =     "M 106.0";
NETWORK
TITLE =
      A     "6S1A";
      AN    "6S1B";
      =     "M 106.1";
NETWORK
TITLE =
      AN    "6S1A";
      A     "6S1B";
      =     "M 106.2";
NETWORK
TITLE =
      AN    "7S1A";
      AN    "7S1B";
      =     "M 107.0";
NETWORK
TITLE =
      A     "7S1A";
      AN    "7S1B";
      =     "M 107.1";
NETWORK
TITLE =
      AN    "7S1A";
      A     "7S1B";
      =     "M 107.2";
NETWORK
TITLE =
      AN    "8S1A";
      AN    "8S1B";
      =     "M 108.0";
NETWORK
TITLE =
      A     "8S1A";
      AN    "8S1B";
      =     "M 108.1";
NETWORK
TITLE =
      AN    "8S1A";
      A     "8S1B";
      =     "M 108.2";
END_FUNCTION

FUNCTION "FC 250" : VOID	// FC 250
VERSION : 0.1
BEGIN
// (block stored without names or comments; labels and parameter names are numbered)
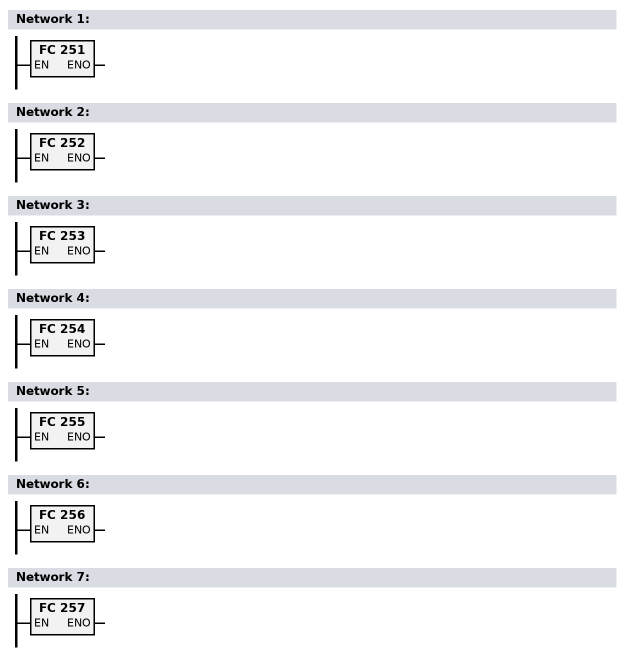
NETWORK
TITLE =
      CALL  "FC 251";
      NOP   0;
NETWORK
TITLE =
      CALL  "FC 252";
      NOP   0;
NETWORK
TITLE =
      CALL  "FC 253";
      NOP   0;
NETWORK
TITLE =
      CALL  "FC 254";
      NOP   0;
NETWORK
TITLE =
      CALL  "FC 255";
      NOP   0;
NETWORK
TITLE =
      CALL  "FC 256";
      NOP   0;
NETWORK
TITLE =
      CALL  "FC 257";
      NOP   0;
END_FUNCTION

FUNCTION "FC 251" : VOID	// FC 251
VERSION : 0.1
BEGIN
// (block stored without names or comments; labels and parameter names are numbered)
